TYPE ST_TARGETS :
STRUCT
	Locomotion_1_target_velocity			AT%Q* : DINT;
	Locomotion_2_target_velocity 			AT%Q* : DINT;
	Locomotion_1_actual_velocity			AT%I* : DINT;
	Locomotion_2_actual_velocity 			AT%I* : DINT;
	Lifter_position_actual_value             AT%I* : DINT;
	Lifter_target_position                     AT%Q* : DINT;
	Rotator_target_position                 AT%Q* : DINT;
	Rotator_position_actual_value             AT%I* : DINT;
	Rotator_target_velocity                 AT%Q* : DINT;
	Rotator_actual_velocity             AT%I* : DINT;
END_STRUCT
END_TYPE

(* stored: Version 1.1.0.1, ProductVersion 3.1.4024.12
   DUT ST_TARGETS: Id {a1ed68a9-c66d-4670-86bc-eac469a31a07} *)
